Staubli VAL3: kill.pgx

public program kill()
begin
  taskKill("tcprec")
end
